PROGRAM MAIN
VAR
	fbMachine			:	FB_Machine(3);
	bButton				:	BOOL;
	bInsertCoin			:	BOOL;
	bTakeProduct		:	BOOL;
	bTakeCoin			:	BOOL;
END_VAR

fbMachine(	bButton	:= bButton,
			bInsertCoin := bInsertCoin,
			bTakeProduct := bTakeProduct,
			bTakeCoin := bTakeCoin);	

bButton := FALSE;
bInsertCoin := FALSE;
bTakeProduct := FALSE;
bTakeCoin := FALSE;

END_PROGRAM

(* stored: Version 1.1.0.1, ProductVersion 3.1.4022.12
   POU MAIN: Id {e0f93eaa-a69b-4cc3-94e8-1fbaf24dd69e}, SpecialFunc None *)
